REGION Network 97: ---
   RUNG wire#powerrail
      Contact( "ON" )
      wire#w1
      Contact( #FB_Enfardadora.EnPaletizadoUT )
      Contact( #Ordenes.TElev_Enfradar )
      wire#w2
      S_Coil( #FB_Enfardadora.ConEnfardadoUT )
   END_RUNG
   RUNG wire#w2
      R_Coil( #FB_Enfardadora.SinEnfardadoUT )
   END_RUNG
   RUNG wire#w1
      I_Contact( #FB_Enfardadora.EnPaletizadoUT )
      wire#w3
      R_Coil( #FB_Enfardadora.ConEnfardadoUT )
   END_RUNG
   RUNG wire#w3
      R_Coil( #FB_Enfardadora.SinEnfardadoUT )
   END_RUNG
   // the same network as SCL:
   IF "ON" AND #FB_Enfardadora.EnPaletizadoUT AND #Ordenes.TElev_Enfradar THEN
       #FB_Enfardadora.ConEnfardadoUT := TRUE;
       #FB_Enfardadora.SinEnfardadoUT := FALSE;
   END_IF;
   IF "ON" AND NOT #FB_Enfardadora.EnPaletizadoUT THEN
       #FB_Enfardadora.ConEnfardadoUT := FALSE;
       #FB_Enfardadora.SinEnfardadoUT := FALSE;
   END_IF;
END_REGION

NETWORK
TITLE = ---
/////////////////////////////////////////////////////////////////////////
// Estado para la Enfardadora

      L     P##EstadoZonaEnfa;  // Puntero a Estado ZONA
      T     #P_EstadoZonaEnfa;

      L     0;  // Inicilizo
      T     LW [#P_EstadoZonaEnfa];

// Automatico - Manual

      A     #EstadoZonaMesa.Automatico_CBx;
      =     #EstadoZonaEnfa.Automatico_CBx;

      A     #EstadoZonaMesa.Manual_CBx;
      =     #EstadoZonaEnfa.Manual_CBx;

// Marcha - Paro - Error

      A     #EstadoZonaMesa.Marcha_CBx;
      =     #EstadoZonaEnfa.Marcha_CBx;

      A     #EstadoZonaMesa.Paro_CBx;
      =     #EstadoZonaEnfa.Paro_CBx;

      A     #EstadoZonaMesa.Error_CBx;
      O     #EstadoZonaMaquina.Error_CBx;
      =     #EstadoZonaEnfa.Error_CBx;

// Reset

      A     #EstadoZonaMesa.Resetear_CBx;
      =     #EstadoZonaEnfa.Resetear_CBx;


REGION Network 99: ---
   RUNG wire#powerrail
      I_Contact( #DesHabilitar_Enfadadora )
      #FB_Enfardadora(CheckElev_EnEnfardadora := wire#w1, EstadoZona := #EstadoZonaEnfa, NDB_Enfardadora := #NDB_Enfardadora, NumMaquina := #MesaElevador, PosicionActual := #PosicionActual, DesHabitar_Enfa := #DesHabilitar_Enfadadora, PorCapas_Enfa := #PorCapas_Enfardado)
   END_RUNG
   RUNG wire#powerrail
      Contact( #CheckElev_EnEnfardadora )
   END_RUNG wire#w1
   RUNG wire#powerrail
      Contact( #ReferenciaOK_Elev )
      { S7_Templates := "SrcType := Int" } LE_Contact(in1 := #PosicionActual, in2 := #PosicionEnfardado)
   END_RUNG wire#w1
   // the same network as SCL:
   IF NOT #DesHabilitar_Enfadadora THEN
       #FB_Enfardadora(EstadoZona := #EstadoZonaEnfa,   // "FB384_Enfardadora_Paletizador_NDD"
                       NDB_Enfardadora := #NDB_Enfardadora,
                       NumMaquina := #MesaElevador,
                       PosicionActual := #PosicionActual,
                       DesHabitar_Enfa := #DesHabilitar_Enfadadora,
                       PorCapas_Enfa := #PorCapas_Enfardado,
                       CheckElev_EnEnfardadora := #CheckElev_EnEnfardadora OR (#ReferenciaOK_Elev AND (#PosicionActual <= #PosicionEnfardado)));
   END_IF;
END_REGION

REGION Network 100: Eventos de Paletizado: Inicio
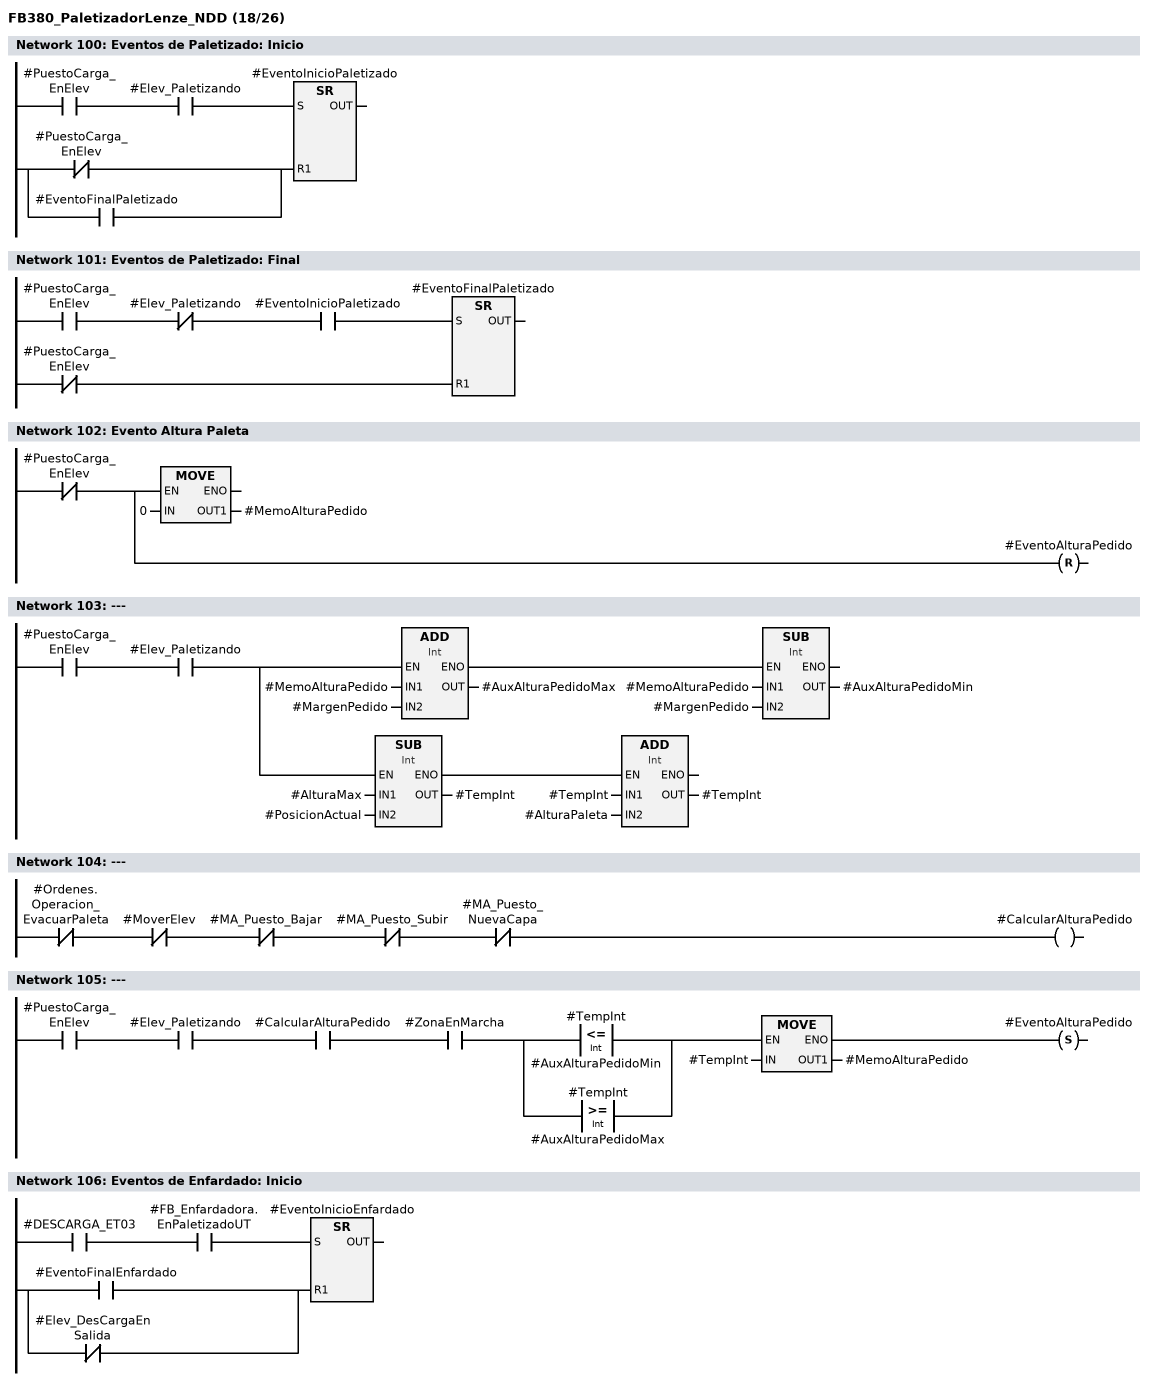
   RUNG wire#powerrail
      Contact( #PuestoCarga_EnElev )
      Contact( #Elev_Paletizando )
      S_SR(operand := #EventoInicioPaletizado, r1 := wire#w1)
   END_RUNG
   RUNG wire#powerrail
      I_Contact( #PuestoCarga_EnElev )
   END_RUNG wire#w1
   RUNG wire#powerrail
      Contact( #EventoFinalPaletizado )
   END_RUNG wire#w1
   // the same network as SCL:
   IF #PuestoCarga_EnElev AND #Elev_Paletizando THEN
       #EventoInicioPaletizado := TRUE;   // SR flip-flop
   END_IF;
   IF NOT #PuestoCarga_EnElev OR #EventoFinalPaletizado THEN #EventoInicioPaletizado := FALSE; END_IF;
END_REGION

REGION Network 101: Eventos de Paletizado: Final
   RUNG wire#powerrail
      Contact( #PuestoCarga_EnElev )
      I_Contact( #Elev_Paletizando )
      Contact( #EventoInicioPaletizado )
      S_SR(operand := #EventoFinalPaletizado, r1 := wire#w1)
   END_RUNG
   RUNG wire#powerrail
      I_Contact( #PuestoCarga_EnElev )
   END_RUNG wire#w1
   // the same network as SCL:
   IF #PuestoCarga_EnElev AND NOT #Elev_Paletizando AND #EventoInicioPaletizado THEN
       #EventoFinalPaletizado := TRUE;   // SR flip-flop
   END_IF;
   IF NOT #PuestoCarga_EnElev THEN #EventoFinalPaletizado := FALSE; END_IF;
END_REGION

REGION Network 102: Evento Altura Paleta
   RUNG wire#powerrail
      I_Contact( #PuestoCarga_EnElev )
      wire#w1
      { S7_GenerateENO := "TRUE" } Move(in := 0, out1 => #MemoAlturaPedido)
   END_RUNG
   RUNG wire#w1
      R_Coil( #EventoAlturaPedido )
   END_RUNG
   // the same network as SCL:
   IF NOT #PuestoCarga_EnElev THEN
       #MemoAlturaPedido := 0;
       #EventoAlturaPedido := FALSE;
   END_IF;
END_REGION

REGION Network 103: ---
   RUNG wire#powerrail
      Contact( #PuestoCarga_EnElev )
      Contact( #Elev_Paletizando )
      wire#w1
      { S7_Templates := "SrcType := Int"; S7_GenerateENO := "TRUE" } Add(in1 := #MemoAlturaPedido, in2 := #MargenPedido, out => #AuxAlturaPedidoMax)
      { S7_Templates := "SrcType := Int"; S7_GenerateENO := "TRUE" } Sub(in1 := #MemoAlturaPedido, in2 := #MargenPedido, out => #AuxAlturaPedidoMin)
   END_RUNG
   RUNG wire#w1
      { S7_Templates := "SrcType := Int"; S7_GenerateENO := "TRUE" } Sub(in1 := #AlturaMax, in2 := #PosicionActual, out => #TempInt)
      { S7_Templates := "SrcType := Int"; S7_GenerateENO := "TRUE" } Add(in1 := #TempInt, in2 := #AlturaPaleta, out => #TempInt)
   END_RUNG
   // the same network as SCL:
   // ENO of a box is taken as its EN; it also drops when the box reports an error
   IF #PuestoCarga_EnElev AND #Elev_Paletizando THEN
       #AuxAlturaPedidoMax := #MemoAlturaPedido + #MargenPedido;
       #AuxAlturaPedidoMin := #MemoAlturaPedido - #MargenPedido;
       #TempInt := #AlturaMax - #PosicionActual;
       #TempInt := #TempInt + #AlturaPaleta;
   END_IF;
END_REGION

REGION Network 104: ---
   RUNG wire#powerrail
      I_Contact( #Ordenes.Operacion_EvacuarPaleta )
      I_Contact( #MoverElev )
      I_Contact( #MA_Puesto_Bajar )
      I_Contact( #MA_Puesto_Subir )
      I_Contact( #MA_Puesto_NuevaCapa )
      Coil( #CalcularAlturaPedido )
   END_RUNG
   // the same network as SCL:
   #CalcularAlturaPedido := NOT #Ordenes.Operacion_EvacuarPaleta AND NOT #MoverElev AND NOT #MA_Puesto_Bajar AND NOT #MA_Puesto_Subir AND NOT #MA_Puesto_NuevaCapa;
END_REGION

REGION Network 105: ---
   RUNG wire#powerrail
      Contact( #PuestoCarga_EnElev )
      Contact( #Elev_Paletizando )
      Contact( #CalcularAlturaPedido )
      Contact( #ZonaEnMarcha )
      wire#w1
      { S7_Templates := "SrcType := Int" } LE_Contact(in1 := #TempInt, in2 := #AuxAlturaPedidoMin)
      wire#w2
      { S7_GenerateENO := "TRUE" } Move(in := #TempInt, out1 => #MemoAlturaPedido)
      S_Coil( #EventoAlturaPedido )
   END_RUNG
   RUNG wire#w1
      { S7_Templates := "SrcType := Int" } GE_Contact(in1 := #TempInt, in2 := #AuxAlturaPedidoMax)
   END_RUNG wire#w2
   // the same network as SCL:
   // ENO of a box is taken as its EN; it also drops when the box reports an error
   IF #PuestoCarga_EnElev AND #Elev_Paletizando AND #CalcularAlturaPedido AND #ZonaEnMarcha AND ((#TempInt <= #AuxAlturaPedidoMin) OR (#TempInt >= #AuxAlturaPedidoMax)) THEN
       #MemoAlturaPedido := #TempInt;
       #EventoAlturaPedido := TRUE;
   END_IF;
END_REGION

REGION Network 106: Eventos de Enfardado: Inicio
   RUNG wire#powerrail
      Contact( #DESCARGA_ET03 )
      Contact( #FB_Enfardadora.EnPaletizadoUT )
      S_SR(operand := #EventoInicioEnfardado, r1 := wire#w1)
   END_RUNG
   RUNG wire#powerrail
      Contact( #EventoFinalEnfardado )
   END_RUNG wire#w1
   RUNG wire#powerrail
      I_Contact( #Elev_DesCargaEnSalida )
   END_RUNG wire#w1
   // the same network as SCL:
   IF #DESCARGA_ET03 AND #FB_Enfardadora.EnPaletizadoUT THEN
       #EventoInicioEnfardado := TRUE;   // SR flip-flop
   END_IF;
   IF #EventoFinalEnfardado OR NOT #Elev_DesCargaEnSalida THEN #EventoInicioEnfardado := FALSE; END_IF;
END_REGION

REGION Network 107: Eventos de Enfardado: Final
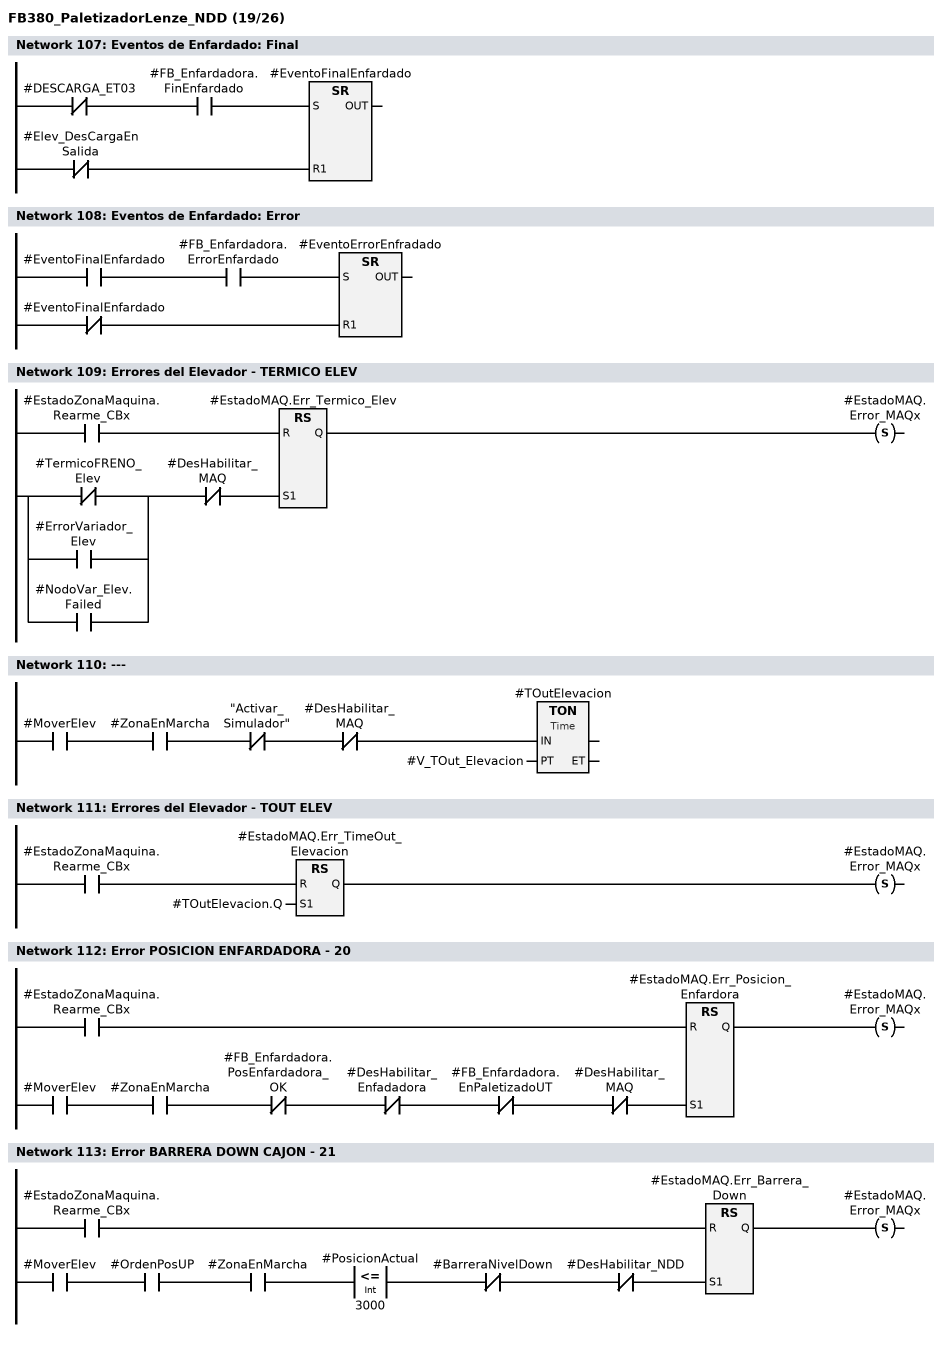
   RUNG wire#powerrail
      I_Contact( #DESCARGA_ET03 )
      Contact( #FB_Enfardadora.FinEnfardado )
      S_SR(operand := #EventoFinalEnfardado, r1 := wire#w1)
   END_RUNG
   RUNG wire#powerrail
      I_Contact( #Elev_DesCargaEnSalida )
   END_RUNG wire#w1
   // the same network as SCL:
   IF NOT #DESCARGA_ET03 AND #FB_Enfardadora.FinEnfardado THEN
       #EventoFinalEnfardado := TRUE;   // SR flip-flop
   END_IF;
   IF NOT #Elev_DesCargaEnSalida THEN #EventoFinalEnfardado := FALSE; END_IF;
END_REGION

REGION Network 108: Eventos de Enfardado: Error
   RUNG wire#powerrail
      Contact( #EventoFinalEnfardado )
      Contact( #FB_Enfardadora.ErrorEnfardado )
      S_SR(operand := #EventoErrorEnfradado, r1 := wire#w1)
   END_RUNG
   RUNG wire#powerrail
      I_Contact( #EventoFinalEnfardado )
   END_RUNG wire#w1
   // the same network as SCL:
   IF #EventoFinalEnfardado AND #FB_Enfardadora.ErrorEnfardado THEN
       #EventoErrorEnfradado := TRUE;   // SR flip-flop
   END_IF;
   IF NOT #EventoFinalEnfardado THEN #EventoErrorEnfradado := FALSE; END_IF;
END_REGION

REGION Network 109: Errores del Elevador - TERMICO ELEV
   RUNG wire#powerrail
      Contact( #EstadoZonaMaquina.Rearme_CBx )
      S_RS(operand := #EstadoMAQ.Err_Termico_Elev, s1 := wire#w2)
      S_Coil( #EstadoMAQ.Error_MAQx )
   END_RUNG
   RUNG wire#powerrail
      I_Contact( #TermicoFRENO_Elev )
      wire#w1
      I_Contact( #DesHabilitar_MAQ )
   END_RUNG wire#w2
   RUNG wire#powerrail
      Contact( #ErrorVariador_Elev )
   END_RUNG wire#w1
   RUNG wire#powerrail
      Contact( #NodoVar_Elev.Failed )
   END_RUNG wire#w1
   // the same network as SCL:
   IF #EstadoZonaMaquina.Rearme_CBx THEN
       #EstadoMAQ.Err_Termico_Elev := FALSE;   // RS flip-flop
   END_IF;
   IF (NOT #TermicoFRENO_Elev OR #ErrorVariador_Elev OR #NodoVar_Elev.Failed) AND NOT #DesHabilitar_MAQ THEN
       #EstadoMAQ.Err_Termico_Elev := TRUE;
   END_IF;
   IF #EstadoMAQ.Err_Termico_Elev THEN #EstadoMAQ.Error_MAQx := TRUE; END_IF;
END_REGION

REGION Network 110: ---
   RUNG wire#powerrail
      Contact( #MoverElev )
      Contact( #ZonaEnMarcha )
      I_Contact( "Activar_Simulador" )
      I_Contact( #DesHabilitar_MAQ )
      { S7_Templates := "time_type := Time" } #TOutElevacion.TON(pt := #V_TOut_Elevacion, et =>)
   END_RUNG
   // the same network as SCL:
   #TOutElevacion(IN := #MoverElev AND #ZonaEnMarcha AND NOT "Activar_Simulador" AND NOT #DesHabilitar_MAQ,   // TON
                  PT := #V_TOut_Elevacion);
END_REGION

REGION Network 111: Errores del Elevador - TOUT ELEV
   RUNG wire#powerrail
      Contact( #EstadoZonaMaquina.Rearme_CBx )
      S_RS(operand := #EstadoMAQ.Err_TimeOut_Elevacion, s1 := #TOutElevacion.Q)
      S_Coil( #EstadoMAQ.Error_MAQx )
   END_RUNG
   // the same network as SCL:
   IF #EstadoZonaMaquina.Rearme_CBx THEN
       #EstadoMAQ.Err_TimeOut_Elevacion := FALSE;   // RS flip-flop
   END_IF;
   IF #TOutElevacion.Q THEN #EstadoMAQ.Err_TimeOut_Elevacion := TRUE; END_IF;
   IF #EstadoMAQ.Err_TimeOut_Elevacion THEN #EstadoMAQ.Error_MAQx := TRUE; END_IF;
END_REGION

REGION Network 112: Error POSICION ENFARDADORA - 20
   RUNG wire#powerrail
      Contact( #EstadoZonaMaquina.Rearme_CBx )
      S_RS(operand := #EstadoMAQ.Err_Posicion_Enfardora, s1 := wire#w1)
      S_Coil( #EstadoMAQ.Error_MAQx )
   END_RUNG
   RUNG wire#powerrail
      Contact( #MoverElev )
      Contact( #ZonaEnMarcha )
      I_Contact( #FB_Enfardadora.PosEnfardadora_OK )
      I_Contact( #DesHabilitar_Enfadadora )
      I_Contact( #FB_Enfardadora.EnPaletizadoUT )
      I_Contact( #DesHabilitar_MAQ )
   END_RUNG wire#w1
   // the same network as SCL:
   IF #EstadoZonaMaquina.Rearme_CBx THEN
       #EstadoMAQ.Err_Posicion_Enfardora := FALSE;   // RS flip-flop
   END_IF;
   IF #MoverElev AND #ZonaEnMarcha AND NOT #FB_Enfardadora.PosEnfardadora_OK AND NOT #DesHabilitar_Enfadadora AND NOT #FB_Enfardadora.EnPaletizadoUT AND NOT #DesHabilitar_MAQ THEN
       #EstadoMAQ.Err_Posicion_Enfardora := TRUE;
   END_IF;
   IF #EstadoMAQ.Err_Posicion_Enfardora THEN #EstadoMAQ.Error_MAQx := TRUE; END_IF;
END_REGION

REGION Network 113: Error BARRERA DOWN CAJON - 21
   RUNG wire#powerrail
      Contact( #EstadoZonaMaquina.Rearme_CBx )
      S_RS(operand := #EstadoMAQ.Err_Barrera_Down, s1 := wire#w1)
      S_Coil( #EstadoMAQ.Error_MAQx )
   END_RUNG
   RUNG wire#powerrail
      Contact( #MoverElev )
      Contact( #OrdenPosUP )
      Contact( #ZonaEnMarcha )
      { S7_Templates := "SrcType := Int" } LE_Contact(in1 := #PosicionActual, in2 := 3000)
      I_Contact( #BarreraNivelDown )
      I_Contact( #DesHabilitar_NDD )
   END_RUNG wire#w1
   // the same network as SCL:
   IF #EstadoZonaMaquina.Rearme_CBx THEN
       #EstadoMAQ.Err_Barrera_Down := FALSE;   // RS flip-flop
   END_IF;
   IF #MoverElev AND #OrdenPosUP AND #ZonaEnMarcha AND (#PosicionActual <= 3000) AND NOT #BarreraNivelDown AND NOT #DesHabilitar_NDD THEN
       #EstadoMAQ.Err_Barrera_Down := TRUE;
   END_IF;
   IF #EstadoMAQ.Err_Barrera_Down THEN #EstadoMAQ.Error_MAQx := TRUE; END_IF;
END_REGION

REGION Network 114: ---
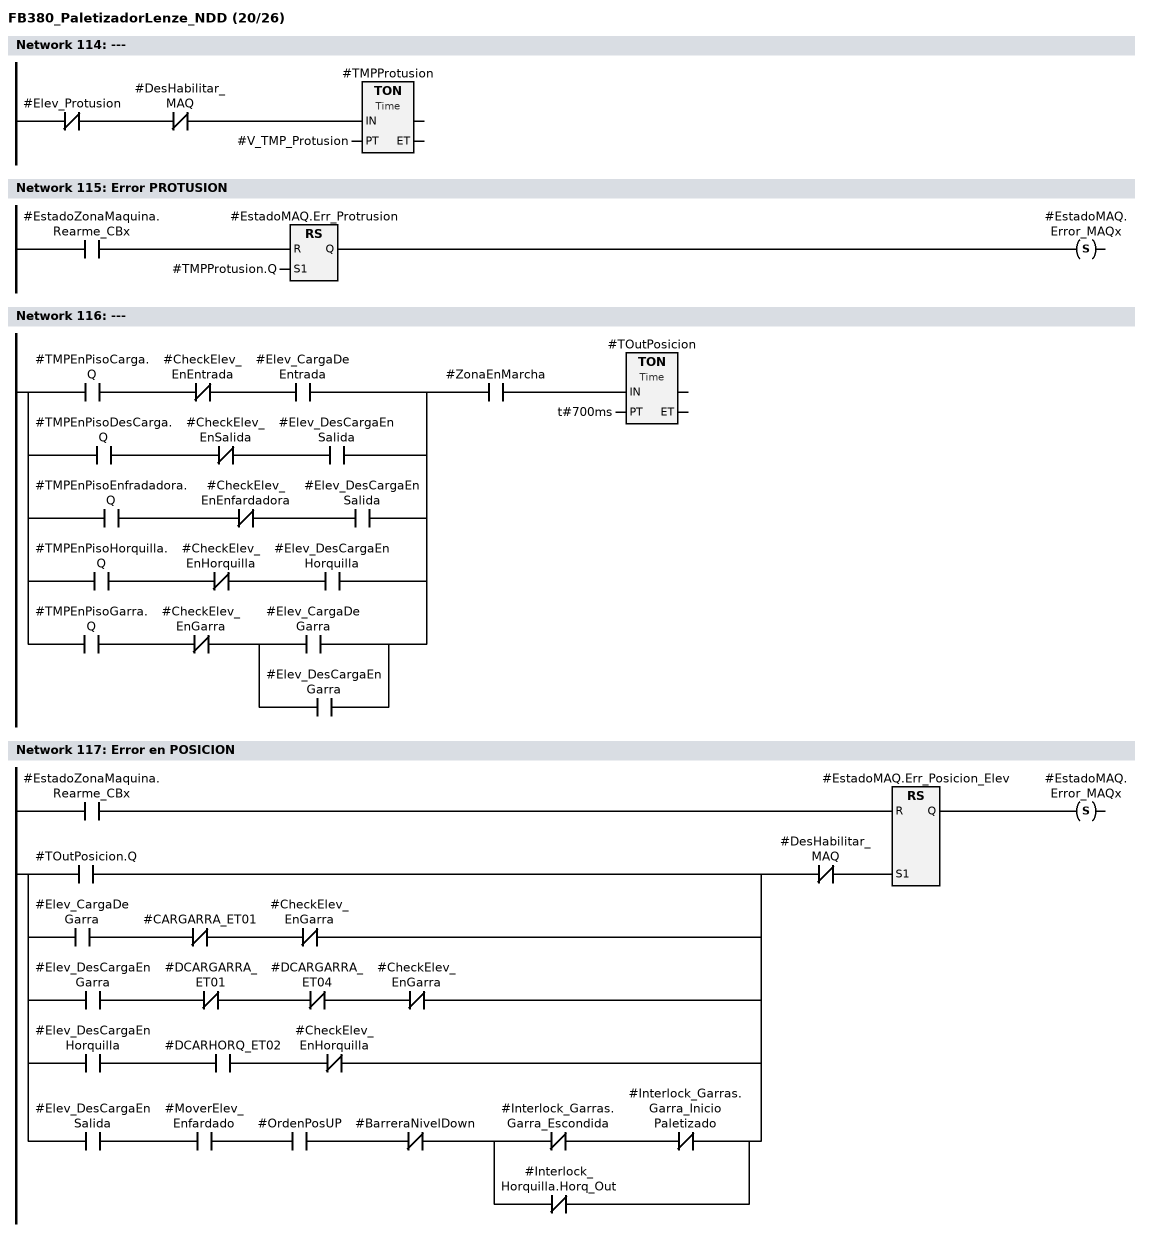
   RUNG wire#powerrail
      I_Contact( #Elev_Protusion )
      I_Contact( #DesHabilitar_MAQ )
      { S7_Templates := "time_type := Time" } #TMPProtusion.TON(pt := #V_TMP_Protusion, et =>)
   END_RUNG
   // the same network as SCL:
   #TMPProtusion(IN := NOT #Elev_Protusion AND NOT #DesHabilitar_MAQ, PT := #V_TMP_Protusion);   // TON
END_REGION

REGION Network 115: Error PROTUSION
   RUNG wire#powerrail
      Contact( #EstadoZonaMaquina.Rearme_CBx )
      S_RS(operand := #EstadoMAQ.Err_Protrusion, s1 := #TMPProtusion.Q)
      S_Coil( #EstadoMAQ.Error_MAQx )
   END_RUNG
   // the same network as SCL:
   IF #EstadoZonaMaquina.Rearme_CBx THEN
       #EstadoMAQ.Err_Protrusion := FALSE;   // RS flip-flop
   END_IF;
   IF #TMPProtusion.Q THEN #EstadoMAQ.Err_Protrusion := TRUE; END_IF;
   IF #EstadoMAQ.Err_Protrusion THEN #EstadoMAQ.Error_MAQx := TRUE; END_IF;
END_REGION

REGION Network 116: ---
   RUNG wire#powerrail
      Contact( #TMPEnPisoCarga.Q )
      I_Contact( #CheckElev_EnEntrada )
      Contact( #Elev_CargaDeEntrada )
      wire#w1
      Contact( #ZonaEnMarcha )
      { S7_Templates := "time_type := Time" } #TOutPosicion.TON(pt := t#700ms, et =>)
   END_RUNG
   RUNG wire#powerrail
      Contact( #TMPEnPisoDesCarga.Q )
      I_Contact( #CheckElev_EnSalida )
      Contact( #Elev_DesCargaEnSalida )
   END_RUNG wire#w1
   RUNG wire#powerrail
      Contact( #TMPEnPisoEnfradadora.Q )
      I_Contact( #CheckElev_EnEnfardadora )
      Contact( #Elev_DesCargaEnSalida )
   END_RUNG wire#w1
   RUNG wire#powerrail
      Contact( #TMPEnPisoHorquilla.Q )
      I_Contact( #CheckElev_EnHorquilla )
      Contact( #Elev_DesCargaEnHorquilla )
   END_RUNG wire#w1
   RUNG wire#powerrail
      Contact( #TMPEnPisoGarra.Q )
      I_Contact( #CheckElev_EnGarra )
      wire#w2
      Contact( #Elev_CargaDeGarra )
   END_RUNG wire#w1
   RUNG wire#w2
      Contact( #Elev_DesCargaEnGarra )
   END_RUNG wire#w1
   // the same network as SCL:
   #TOutPosicion(IN := ((#TMPEnPisoCarga.Q AND NOT #CheckElev_EnEntrada AND #Elev_CargaDeEntrada) OR (#TMPEnPisoDesCarga.Q AND NOT #CheckElev_EnSalida AND #Elev_DesCargaEnSalida) OR (#TMPEnPisoEnfradadora.Q AND NOT #CheckElev_EnEnfardadora AND #Elev_DesCargaEnSalida) OR (#TMPEnPisoHorquilla.Q AND NOT #CheckElev_EnHorquilla AND #Elev_DesCargaEnHorquilla) OR (#TMPEnPisoGarra.Q AND NOT #CheckElev_EnGarra AND (#Elev_CargaDeGarra OR #Elev_DesCargaEnGarra))) AND #ZonaEnMarcha,   // TON
                 PT := t#700ms);
END_REGION

REGION Network 117: Error en POSICION
   RUNG wire#powerrail
      Contact( #EstadoZonaMaquina.Rearme_CBx )
      S_RS(operand := #EstadoMAQ.Err_Posicion_Elev, s1 := wire#w3)
      S_Coil( #EstadoMAQ.Error_MAQx )
   END_RUNG
   RUNG wire#powerrail
      Contact( #TOutPosicion.Q )
      wire#w1
      I_Contact( #DesHabilitar_MAQ )
   END_RUNG wire#w3
   RUNG wire#powerrail
      Contact( #Elev_CargaDeGarra )
      I_Contact( #CARGARRA_ET01 )
      I_Contact( #CheckElev_EnGarra )
   END_RUNG wire#w1
   RUNG wire#powerrail
      Contact( #Elev_DesCargaEnGarra )
      I_Contact( #DCARGARRA_ET01 )
      I_Contact( #DCARGARRA_ET04 )
      I_Contact( #CheckElev_EnGarra )
   END_RUNG wire#w1
   RUNG wire#powerrail
      Contact( #Elev_DesCargaEnHorquilla )
      Contact( #DCARHORQ_ET02 )
      I_Contact( #CheckElev_EnHorquilla )
   END_RUNG wire#w1
   RUNG wire#powerrail
      Contact( #Elev_DesCargaEnSalida )
      Contact( #MoverElev_Enfardado )
      Contact( #OrdenPosUP )
      I_Contact( #BarreraNivelDown )
      wire#w2
      I_Contact( #Interlock_Garras.Garra_Escondida )
      I_Contact( #Interlock_Garras.Garra_InicioPaletizado )
   END_RUNG wire#w1
   RUNG wire#w2
      I_Contact( #Interlock_Horquilla.Horq_Out )
   END_RUNG wire#w1
   // the same network as SCL:
   IF #EstadoZonaMaquina.Rearme_CBx THEN
       #EstadoMAQ.Err_Posicion_Elev := FALSE;   // RS flip-flop
   END_IF;
   IF (#TOutPosicion.Q OR (#Elev_CargaDeGarra AND NOT #CARGARRA_ET01 AND NOT #CheckElev_EnGarra) OR (#Elev_DesCargaEnGarra AND NOT #DCARGARRA_ET01 AND NOT #DCARGARRA_ET04 AND NOT #CheckElev_EnGarra) OR (#Elev_DesCargaEnHorquilla AND #DCARHORQ_ET02 AND NOT #CheckElev_EnHorquilla) OR (#Elev_DesCargaEnSalida AND #MoverElev_Enfardado AND #OrdenPosUP AND NOT #BarreraNivelDown AND ((NOT #Interlock_Garras.Garra_Escondida AND NOT #Interlock_Garras.Garra_InicioPaletizado) OR NOT #Interlock_Horquilla.Horq_Out))) AND NOT #DesHabilitar_MAQ THEN
       #EstadoMAQ.Err_Posicion_Elev := TRUE;
   END_IF;
   IF #EstadoMAQ.Err_Posicion_Elev THEN #EstadoMAQ.Error_MAQx := TRUE; END_IF;
END_REGION

REGION Network 118: Error REFERENCIA ELEV - 5
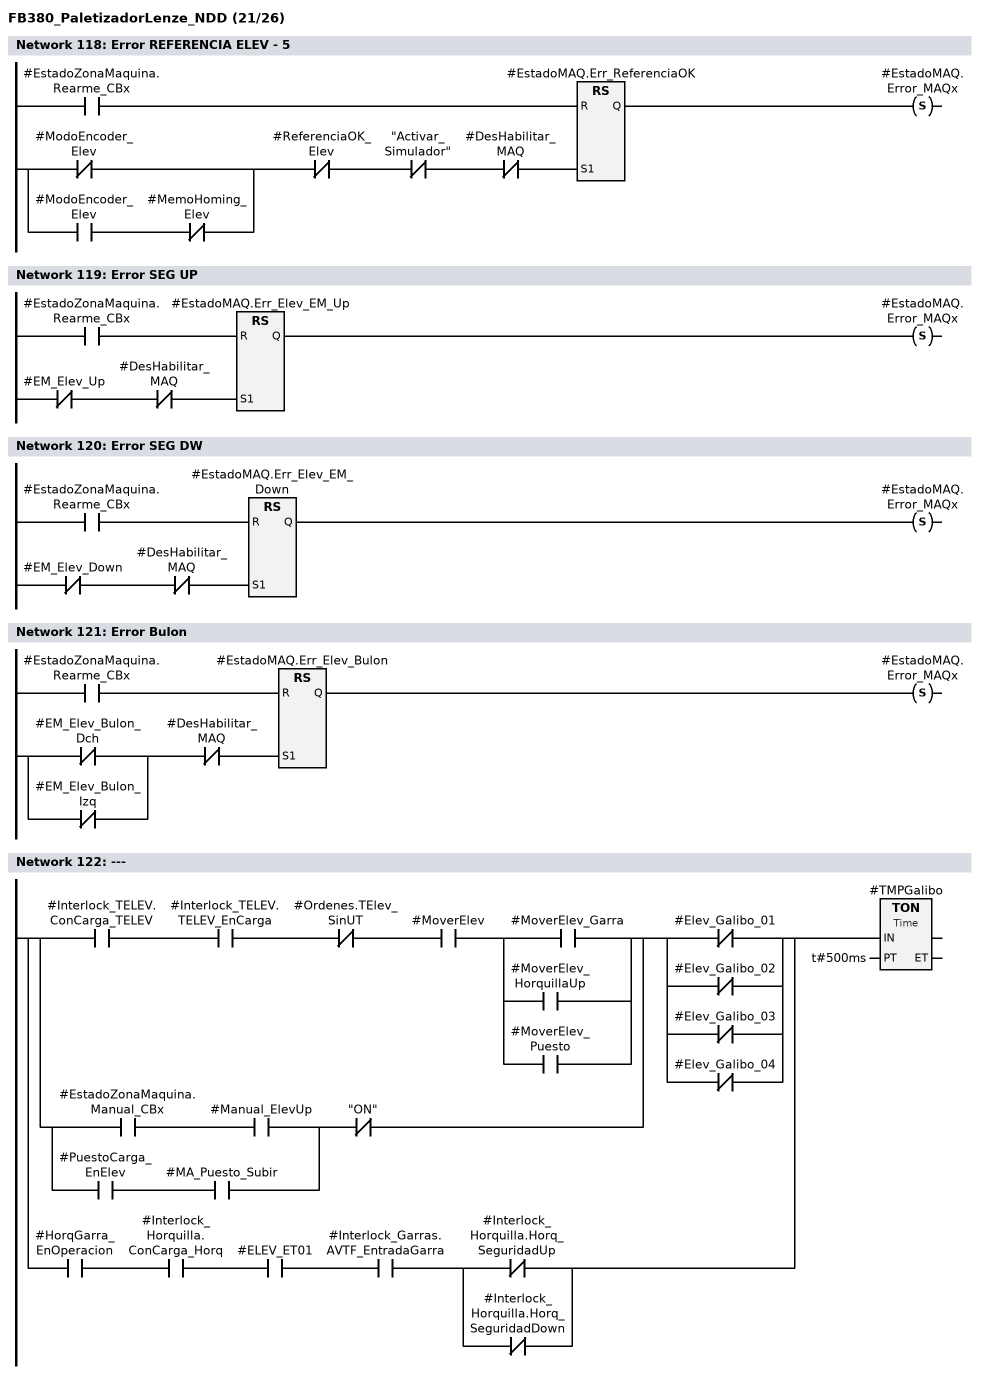
   RUNG wire#powerrail
      Contact( #EstadoZonaMaquina.Rearme_CBx )
      S_RS(operand := #EstadoMAQ.Err_ReferenciaOK, s1 := wire#w2)
      S_Coil( #EstadoMAQ.Error_MAQx )
   END_RUNG
   RUNG wire#powerrail
      I_Contact( #ModoEncoder_Elev )
      wire#w1
      I_Contact( #ReferenciaOK_Elev )
      I_Contact( "Activar_Simulador" )
      I_Contact( #DesHabilitar_MAQ )
   END_RUNG wire#w2
   RUNG wire#powerrail
      Contact( #ModoEncoder_Elev )
      I_Contact( #MemoHoming_Elev )
   END_RUNG wire#w1
   // the same network as SCL:
   IF #EstadoZonaMaquina.Rearme_CBx THEN
       #EstadoMAQ.Err_ReferenciaOK := FALSE;   // RS flip-flop
   END_IF;
   IF (NOT #ModoEncoder_Elev OR (#ModoEncoder_Elev AND NOT #MemoHoming_Elev)) AND NOT #ReferenciaOK_Elev AND NOT "Activar_Simulador" AND NOT #DesHabilitar_MAQ THEN
       #EstadoMAQ.Err_ReferenciaOK := TRUE;
   END_IF;
   IF #EstadoMAQ.Err_ReferenciaOK THEN #EstadoMAQ.Error_MAQx := TRUE; END_IF;
END_REGION

REGION Network 119: Error SEG UP
   RUNG wire#powerrail
      Contact( #EstadoZonaMaquina.Rearme_CBx )
      S_RS(operand := #EstadoMAQ.Err_Elev_EM_Up, s1 := wire#w1)
      S_Coil( #EstadoMAQ.Error_MAQx )
   END_RUNG
   RUNG wire#powerrail
      I_Contact( #EM_Elev_Up )
      I_Contact( #DesHabilitar_MAQ )
   END_RUNG wire#w1
   // the same network as SCL:
   IF #EstadoZonaMaquina.Rearme_CBx THEN
       #EstadoMAQ.Err_Elev_EM_Up := FALSE;   // RS flip-flop
   END_IF;
   IF NOT #EM_Elev_Up AND NOT #DesHabilitar_MAQ THEN #EstadoMAQ.Err_Elev_EM_Up := TRUE; END_IF;
   IF #EstadoMAQ.Err_Elev_EM_Up THEN #EstadoMAQ.Error_MAQx := TRUE; END_IF;
END_REGION

REGION Network 120: Error SEG DW
   RUNG wire#powerrail
      Contact( #EstadoZonaMaquina.Rearme_CBx )
      S_RS(operand := #EstadoMAQ.Err_Elev_EM_Down, s1 := wire#w1)
      S_Coil( #EstadoMAQ.Error_MAQx )
   END_RUNG
   RUNG wire#powerrail
      I_Contact( #EM_Elev_Down )
      I_Contact( #DesHabilitar_MAQ )
   END_RUNG wire#w1
   // the same network as SCL:
   IF #EstadoZonaMaquina.Rearme_CBx THEN
       #EstadoMAQ.Err_Elev_EM_Down := FALSE;   // RS flip-flop
   END_IF;
   IF NOT #EM_Elev_Down AND NOT #DesHabilitar_MAQ THEN #EstadoMAQ.Err_Elev_EM_Down := TRUE; END_IF;
   IF #EstadoMAQ.Err_Elev_EM_Down THEN #EstadoMAQ.Error_MAQx := TRUE; END_IF;
END_REGION

REGION Network 121: Error Bulon
   RUNG wire#powerrail
      Contact( #EstadoZonaMaquina.Rearme_CBx )
      S_RS(operand := #EstadoMAQ.Err_Elev_Bulon, s1 := wire#w2)
      S_Coil( #EstadoMAQ.Error_MAQx )
   END_RUNG
   RUNG wire#powerrail
      I_Contact( #EM_Elev_Bulon_Dch )
      wire#w1
      I_Contact( #DesHabilitar_MAQ )
   END_RUNG wire#w2
   RUNG wire#powerrail
      I_Contact( #EM_Elev_Bulon_Izq )
   END_RUNG wire#w1
   // the same network as SCL:
   IF #EstadoZonaMaquina.Rearme_CBx THEN
       #EstadoMAQ.Err_Elev_Bulon := FALSE;   // RS flip-flop
   END_IF;
   IF (NOT #EM_Elev_Bulon_Dch OR NOT #EM_Elev_Bulon_Izq) AND NOT #DesHabilitar_MAQ THEN
       #EstadoMAQ.Err_Elev_Bulon := TRUE;
   END_IF;
   IF #EstadoMAQ.Err_Elev_Bulon THEN #EstadoMAQ.Error_MAQx := TRUE; END_IF;
END_REGION

REGION Network 122: ---
   RUNG wire#powerrail
      Contact( #Interlock_TELEV.ConCarga_TELEV )
      Contact( #Interlock_TELEV.TELEV_EnCarga )
      I_Contact( #Ordenes.TElev_SinUT )
      Contact( #MoverElev )
      wire#w1
      Contact( #MoverElev_Garra )
      wire#w2
      I_Contact( #Elev_Galibo_01 )
      wire#w4
      { S7_Templates := "time_type := Time" } #TMPGalibo.TON(pt := t#500ms, et =>)
   END_RUNG
   RUNG wire#w1
      Contact( #MoverElev_HorquillaUp )
   END_RUNG wire#w2
   RUNG wire#w1
      Contact( #MoverElev_Puesto )
   END_RUNG wire#w2
   RUNG wire#powerrail
      Contact( #EstadoZonaMaquina.Manual_CBx )
      Contact( #Manual_ElevUp )
      wire#w3
      I_Contact( "ON" )
   END_RUNG wire#w2
   RUNG wire#powerrail
      Contact( #PuestoCarga_EnElev )
      Contact( #MA_Puesto_Subir )
   END_RUNG wire#w3
   RUNG wire#w2
      I_Contact( #Elev_Galibo_02 )
   END_RUNG wire#w4
   RUNG wire#w2
      I_Contact( #Elev_Galibo_03 )
   END_RUNG wire#w4
   RUNG wire#w2
      I_Contact( #Elev_Galibo_04 )
   END_RUNG wire#w4
   RUNG wire#powerrail
      Contact( #HorqGarra_EnOperacion )
      Contact( #Interlock_Horquilla.ConCarga_Horq )
      Contact( #ELEV_ET01 )
      Contact( #Interlock_Garras.AVTF_EntradaGarra )
      wire#w5
      I_Contact( #Interlock_Horquilla.Horq_SeguridadUp )
   END_RUNG wire#w4
   RUNG wire#w5
      I_Contact( #Interlock_Horquilla.Horq_SeguridadDown )
   END_RUNG wire#w4
   // the same network as SCL:
   #TMPGalibo(IN := (((#Interlock_TELEV.ConCarga_TELEV AND #Interlock_TELEV.TELEV_EnCarga AND NOT #Ordenes.TElev_SinUT AND #MoverElev AND (#MoverElev_Garra OR #MoverElev_HorquillaUp OR #MoverElev_Puesto)) OR (((#EstadoZonaMaquina.Manual_CBx AND #Manual_ElevUp) OR (#PuestoCarga_EnElev AND #MA_Puesto_Subir)) AND NOT "ON")) AND (NOT #Elev_Galibo_01 OR NOT #Elev_Galibo_02 OR NOT #Elev_Galibo_03 OR NOT #Elev_Galibo_04)) OR (#HorqGarra_EnOperacion AND #Interlock_Horquilla.ConCarga_Horq AND #ELEV_ET01 AND #Interlock_Garras.AVTF_EntradaGarra AND (NOT #Interlock_Horquilla.Horq_SeguridadUp OR NOT #Interlock_Horquilla.Horq_SeguridadDown)),   // TON
              PT := t#500ms);
END_REGION

REGION Network 123: Error PHS GALIBO
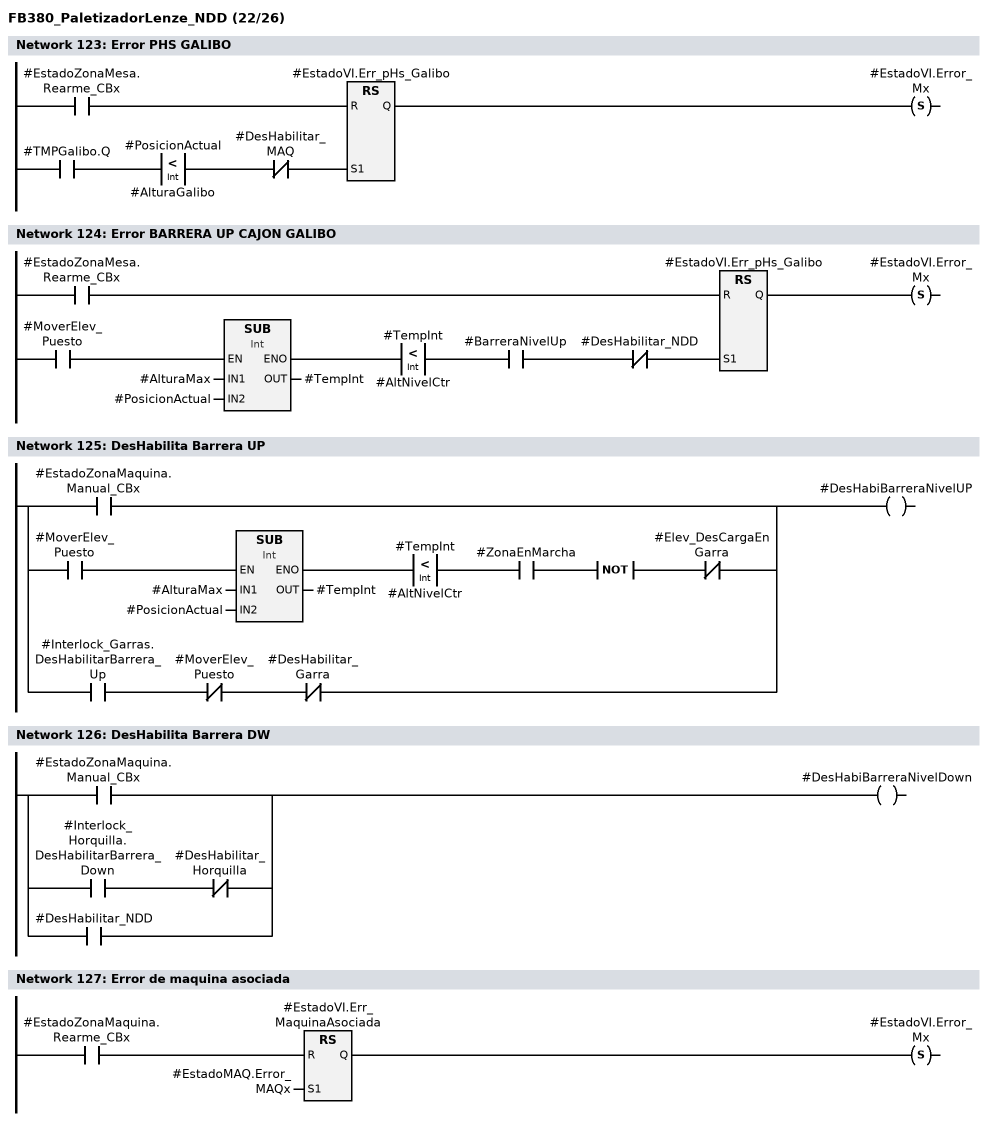
   RUNG wire#powerrail
      Contact( #EstadoZonaMesa.Rearme_CBx )
      S_RS(operand := #EstadoVI.Err_pHs_Galibo, s1 := wire#w1)
      S_Coil( #EstadoVI.Error_Mx )
   END_RUNG
   RUNG wire#powerrail
      Contact( #TMPGalibo.Q )
      { S7_Templates := "SrcType := Int" } LT_Contact(in1 := #PosicionActual, in2 := #AlturaGalibo)
      I_Contact( #DesHabilitar_MAQ )
   END_RUNG wire#w1
   // the same network as SCL:
   IF #EstadoZonaMesa.Rearme_CBx THEN
       #EstadoVI.Err_pHs_Galibo := FALSE;   // RS flip-flop
   END_IF;
   IF #TMPGalibo.Q AND (#PosicionActual < #AlturaGalibo) AND NOT #DesHabilitar_MAQ THEN
       #EstadoVI.Err_pHs_Galibo := TRUE;
   END_IF;
   IF #EstadoVI.Err_pHs_Galibo THEN #EstadoVI.Error_Mx := TRUE; END_IF;
END_REGION

REGION Network 124: Error BARRERA UP CAJON GALIBO
   RUNG wire#powerrail
      Contact( #EstadoZonaMesa.Rearme_CBx )
      S_RS(operand := #EstadoVI.Err_pHs_Galibo, s1 := wire#w1)
      S_Coil( #EstadoVI.Error_Mx )
   END_RUNG
   RUNG wire#powerrail
      Contact( #MoverElev_Puesto )
      { S7_Templates := "SrcType := Int"; S7_GenerateENO := "TRUE" } Sub(in1 := #AlturaMax, in2 := #PosicionActual, out => #TempInt)
      { S7_Templates := "SrcType := Int" } LT_Contact(in1 := #TempInt, in2 := #AltNivelCtr)
      Contact( #BarreraNivelUp )
      I_Contact( #DesHabilitar_NDD )
   END_RUNG wire#w1
   // the same network as SCL:
   // ENO of a box is taken as its EN; it also drops when the box reports an error
   IF #MoverElev_Puesto THEN #TempInt := #AlturaMax - #PosicionActual; END_IF;
   IF #EstadoZonaMesa.Rearme_CBx THEN
       #EstadoVI.Err_pHs_Galibo := FALSE;   // RS flip-flop
   END_IF;
   IF #MoverElev_Puesto AND (#TempInt < #AltNivelCtr) AND #BarreraNivelUp AND NOT #DesHabilitar_NDD THEN
       #EstadoVI.Err_pHs_Galibo := TRUE;
   END_IF;
   IF #EstadoVI.Err_pHs_Galibo THEN #EstadoVI.Error_Mx := TRUE; END_IF;
END_REGION

REGION Network 125: DesHabilita Barrera UP
   RUNG wire#powerrail
      Contact( #EstadoZonaMaquina.Manual_CBx )
      wire#w1
      Coil( #DesHabiBarreraNivelUP )
   END_RUNG
   RUNG wire#powerrail
      Contact( #MoverElev_Puesto )
      { S7_Templates := "SrcType := Int"; S7_GenerateENO := "TRUE" } Sub(in1 := #AlturaMax, in2 := #PosicionActual, out => #TempInt)
      { S7_Templates := "SrcType := Int" } LT_Contact(in1 := #TempInt, in2 := #AltNivelCtr)
      Contact( #ZonaEnMarcha )
      Not()
      I_Contact( #Elev_DesCargaEnGarra )
   END_RUNG wire#w1
   RUNG wire#powerrail
      Contact( #Interlock_Garras.DesHabilitarBarrera_Up )
      I_Contact( #MoverElev_Puesto )
      I_Contact( #DesHabilitar_Garra )
   END_RUNG wire#w1
   // the same network as SCL:
   // ENO of a box is taken as its EN; it also drops when the box reports an error
   IF #MoverElev_Puesto THEN #TempInt := #AlturaMax - #PosicionActual; END_IF;
   #DesHabiBarreraNivelUP := #EstadoZonaMaquina.Manual_CBx OR (NOT (#MoverElev_Puesto AND (#TempInt < #AltNivelCtr) AND #ZonaEnMarcha) AND NOT #Elev_DesCargaEnGarra) OR (#Interlock_Garras.DesHabilitarBarrera_Up AND NOT #MoverElev_Puesto AND NOT #DesHabilitar_Garra);
END_REGION

REGION Network 126: DesHabilita Barrera DW
   RUNG wire#powerrail
      Contact( #EstadoZonaMaquina.Manual_CBx )
      wire#w1
      Coil( #DesHabiBarreraNivelDown )
   END_RUNG
   RUNG wire#powerrail
      Contact( #Interlock_Horquilla.DesHabilitarBarrera_Down )
      I_Contact( #DesHabilitar_Horquilla )
   END_RUNG wire#w1
   RUNG wire#powerrail
      Contact( #DesHabilitar_NDD )
   END_RUNG wire#w1
   // the same network as SCL:
   #DesHabiBarreraNivelDown := #EstadoZonaMaquina.Manual_CBx OR (#Interlock_Horquilla.DesHabilitarBarrera_Down AND NOT #DesHabilitar_Horquilla) OR #DesHabilitar_NDD;
END_REGION

REGION Network 127: Error de maquina asociada
   RUNG wire#powerrail
      Contact( #EstadoZonaMaquina.Rearme_CBx )
      S_RS(operand := #EstadoVI.Err_MaquinaAsociada, s1 := #EstadoMAQ.Error_MAQx)
      S_Coil( #EstadoVI.Error_Mx )
   END_RUNG
   // the same network as SCL:
   IF #EstadoZonaMaquina.Rearme_CBx THEN
       #EstadoVI.Err_MaquinaAsociada := FALSE;   // RS flip-flop
   END_IF;
   IF #EstadoMAQ.Error_MAQx THEN #EstadoVI.Err_MaquinaAsociada := TRUE; END_IF;
   IF #EstadoVI.Err_MaquinaAsociada THEN #EstadoVI.Error_Mx := TRUE; END_IF;
END_REGION

REGION Network 128: Estado del Elevador
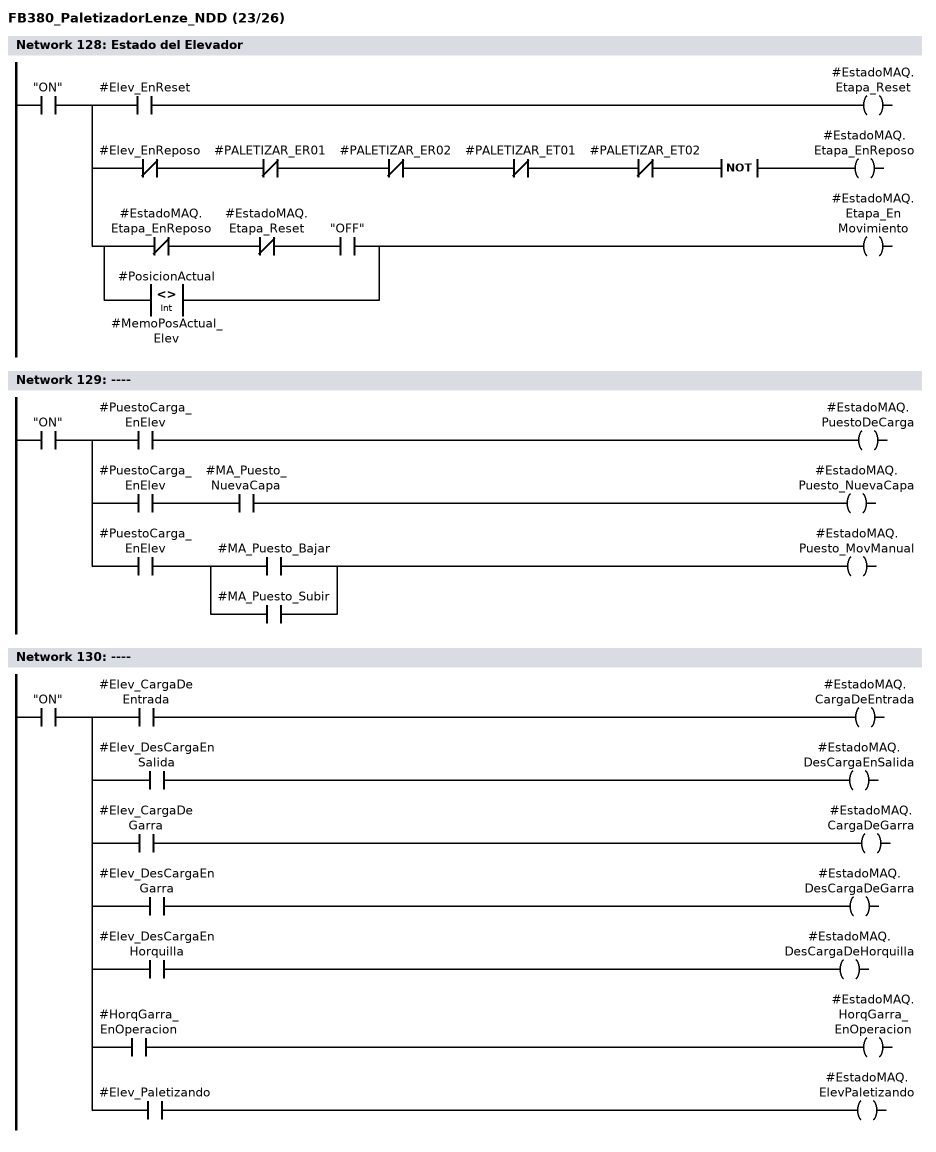
   RUNG wire#powerrail
      Contact( "ON" )
      wire#w1
      Contact( #Elev_EnReset )
      Coil( #EstadoMAQ.Etapa_Reset )
   END_RUNG
   RUNG wire#w1
      I_Contact( #Elev_EnReposo )
      I_Contact( #PALETIZAR_ER01 )
      I_Contact( #PALETIZAR_ER02 )
      I_Contact( #PALETIZAR_ET01 )
      I_Contact( #PALETIZAR_ET02 )
      Not()
      Coil( #EstadoMAQ.Etapa_EnReposo )
   END_RUNG
   RUNG wire#w1
      I_Contact( #EstadoMAQ.Etapa_EnReposo )
      I_Contact( #EstadoMAQ.Etapa_Reset )
      Contact( "OFF" )
      wire#w2
      Coil( #EstadoMAQ.Etapa_EnMovimiento )
   END_RUNG
   RUNG wire#w1
      { S7_Templates := "SrcType := Int" } NE_Contact(in1 := #PosicionActual, in2 := #MemoPosActual_Elev)
   END_RUNG wire#w2
   // the same network as SCL:
   #EstadoMAQ.Etapa_Reset := "ON" AND #Elev_EnReset;
   #EstadoMAQ.Etapa_EnReposo := NOT ("ON" AND NOT #Elev_EnReposo AND NOT #PALETIZAR_ER01 AND NOT #PALETIZAR_ER02 AND NOT #PALETIZAR_ET01 AND NOT #PALETIZAR_ET02);
   #EstadoMAQ.Etapa_EnMovimiento := "ON" AND ((NOT #EstadoMAQ.Etapa_EnReposo AND NOT #EstadoMAQ.Etapa_Reset AND "OFF") OR (#PosicionActual <> #MemoPosActual_Elev));
END_REGION

REGION Network 129: ----
   RUNG wire#powerrail
      Contact( "ON" )
      wire#w1
      Contact( #PuestoCarga_EnElev )
      Coil( #EstadoMAQ.PuestoDeCarga )
   END_RUNG
   RUNG wire#w1
      Contact( #PuestoCarga_EnElev )
      Contact( #MA_Puesto_NuevaCapa )
      Coil( #EstadoMAQ.Puesto_NuevaCapa )
   END_RUNG
   RUNG wire#w1
      Contact( #PuestoCarga_EnElev )
      wire#w2
      Contact( #MA_Puesto_Bajar )
      wire#w3
      Coil( #EstadoMAQ.Puesto_MovManual )
   END_RUNG
   RUNG wire#w2
      Contact( #MA_Puesto_Subir )
   END_RUNG wire#w3
   // the same network as SCL:
   #EstadoMAQ.PuestoDeCarga := "ON" AND #PuestoCarga_EnElev;
   #EstadoMAQ.Puesto_NuevaCapa := "ON" AND #PuestoCarga_EnElev AND #MA_Puesto_NuevaCapa;
   #EstadoMAQ.Puesto_MovManual := "ON" AND #PuestoCarga_EnElev AND (#MA_Puesto_Bajar OR #MA_Puesto_Subir);
END_REGION

REGION Network 130: ----
   RUNG wire#powerrail
      Contact( "ON" )
      wire#w1
      Contact( #Elev_CargaDeEntrada )
      Coil( #EstadoMAQ.CargaDeEntrada )
   END_RUNG
   RUNG wire#w1
      Contact( #Elev_DesCargaEnSalida )
      Coil( #EstadoMAQ.DesCargaEnSalida )
   END_RUNG
   RUNG wire#w1
      Contact( #Elev_CargaDeGarra )
      Coil( #EstadoMAQ.CargaDeGarra )
   END_RUNG
   RUNG wire#w1
      Contact( #Elev_DesCargaEnGarra )
      Coil( #EstadoMAQ.DesCargaDeGarra )
   END_RUNG
   RUNG wire#w1
      Contact( #Elev_DesCargaEnHorquilla )
      Coil( #EstadoMAQ.DesCargaDeHorquilla )
   END_RUNG
   RUNG wire#w1
      Contact( #HorqGarra_EnOperacion )
      Coil( #EstadoMAQ.HorqGarra_EnOperacion )
   END_RUNG
   RUNG wire#w1
      Contact( #Elev_Paletizando )
      Coil( #EstadoMAQ.ElevPaletizando )
   END_RUNG
   // the same network as SCL:
   #EstadoMAQ.CargaDeEntrada := "ON" AND #Elev_CargaDeEntrada;
   #EstadoMAQ.DesCargaEnSalida := "ON" AND #Elev_DesCargaEnSalida;
   #EstadoMAQ.CargaDeGarra := "ON" AND #Elev_CargaDeGarra;
   #EstadoMAQ.DesCargaDeGarra := "ON" AND #Elev_DesCargaEnGarra;
   #EstadoMAQ.DesCargaDeHorquilla := "ON" AND #Elev_DesCargaEnHorquilla;
   #EstadoMAQ.HorqGarra_EnOperacion := "ON" AND #HorqGarra_EnOperacion;
   #EstadoMAQ.ElevPaletizando := "ON" AND #Elev_Paletizando;
END_REGION

REGION Network 131: Entradas del Elevador
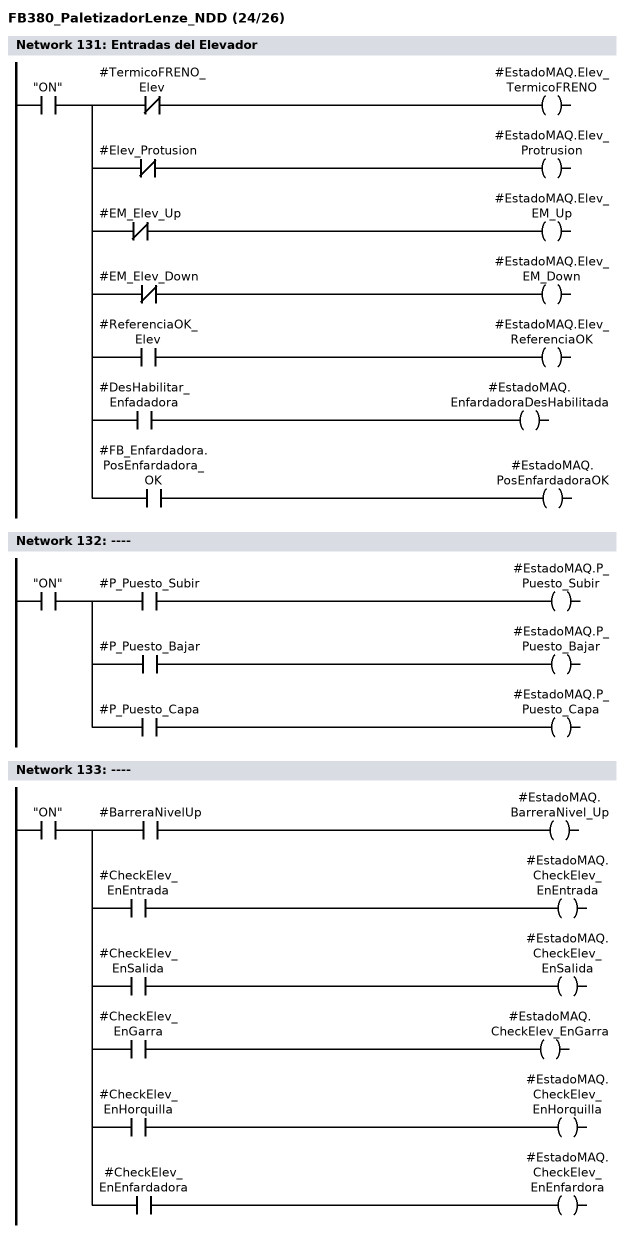
   RUNG wire#powerrail
      Contact( "ON" )
      wire#w1
      I_Contact( #TermicoFRENO_Elev )
      Coil( #EstadoMAQ.Elev_TermicoFRENO )
   END_RUNG
   RUNG wire#w1
      I_Contact( #Elev_Protusion )
      Coil( #EstadoMAQ.Elev_Protrusion )
   END_RUNG
   RUNG wire#w1
      I_Contact( #EM_Elev_Up )
      Coil( #EstadoMAQ.Elev_EM_Up )
   END_RUNG
   RUNG wire#w1
      I_Contact( #EM_Elev_Down )
      Coil( #EstadoMAQ.Elev_EM_Down )
   END_RUNG
   RUNG wire#w1
      Contact( #ReferenciaOK_Elev )
      Coil( #EstadoMAQ.Elev_ReferenciaOK )
   END_RUNG
   RUNG wire#w1
      Contact( #DesHabilitar_Enfadadora )
      Coil( #EstadoMAQ.EnfardadoraDesHabilitada )
   END_RUNG
   RUNG wire#w1
      Contact( #FB_Enfardadora.PosEnfardadora_OK )
      Coil( #EstadoMAQ.PosEnfardadoraOK )
   END_RUNG
   // the same network as SCL:
   #EstadoMAQ.Elev_TermicoFRENO := "ON" AND NOT #TermicoFRENO_Elev;
   #EstadoMAQ.Elev_Protrusion := "ON" AND NOT #Elev_Protusion;
   #EstadoMAQ.Elev_EM_Up := "ON" AND NOT #EM_Elev_Up;
   #EstadoMAQ.Elev_EM_Down := "ON" AND NOT #EM_Elev_Down;
   #EstadoMAQ.Elev_ReferenciaOK := "ON" AND #ReferenciaOK_Elev;
   #EstadoMAQ.EnfardadoraDesHabilitada := "ON" AND #DesHabilitar_Enfadadora;
   #EstadoMAQ.PosEnfardadoraOK := "ON" AND #FB_Enfardadora.PosEnfardadora_OK;
END_REGION

REGION Network 132: ----
   RUNG wire#powerrail
      Contact( "ON" )
      wire#w1
      Contact( #P_Puesto_Subir )
      Coil( #EstadoMAQ.P_Puesto_Subir )
   END_RUNG
   RUNG wire#w1
      Contact( #P_Puesto_Bajar )
      Coil( #EstadoMAQ.P_Puesto_Bajar )
   END_RUNG
   RUNG wire#w1
      Contact( #P_Puesto_Capa )
      Coil( #EstadoMAQ.P_Puesto_Capa )
   END_RUNG
   // the same network as SCL:
   #EstadoMAQ.P_Puesto_Subir := "ON" AND #P_Puesto_Subir;
   #EstadoMAQ.P_Puesto_Bajar := "ON" AND #P_Puesto_Bajar;
   #EstadoMAQ.P_Puesto_Capa := "ON" AND #P_Puesto_Capa;
END_REGION

REGION Network 133: ----
   RUNG wire#powerrail
      Contact( "ON" )
      wire#w1
      Contact( #BarreraNivelUp )
      Coil( #EstadoMAQ.BarreraNivel_Up )
   END_RUNG
   RUNG wire#w1
      Contact( #CheckElev_EnEntrada )
      Coil( #EstadoMAQ.CheckElev_EnEntrada )
   END_RUNG
   RUNG wire#w1
      Contact( #CheckElev_EnSalida )
      Coil( #EstadoMAQ.CheckElev_EnSalida )
   END_RUNG
   RUNG wire#w1
      Contact( #CheckElev_EnGarra )
      Coil( #EstadoMAQ.CheckElev_EnGarra )
   END_RUNG
   RUNG wire#w1
      Contact( #CheckElev_EnHorquilla )
      Coil( #EstadoMAQ.CheckElev_EnHorquilla )
   END_RUNG
   RUNG wire#w1
      Contact( #CheckElev_EnEnfardadora )
      Coil( #EstadoMAQ.CheckElev_EnEnfardora )
   END_RUNG
   // the same network as SCL:
   #EstadoMAQ.BarreraNivel_Up := "ON" AND #BarreraNivelUp;
   #EstadoMAQ.CheckElev_EnEntrada := "ON" AND #CheckElev_EnEntrada;
   #EstadoMAQ.CheckElev_EnSalida := "ON" AND #CheckElev_EnSalida;
   #EstadoMAQ.CheckElev_EnGarra := "ON" AND #CheckElev_EnGarra;
   #EstadoMAQ.CheckElev_EnHorquilla := "ON" AND #CheckElev_EnHorquilla;
   #EstadoMAQ.CheckElev_EnEnfardora := "ON" AND #CheckElev_EnEnfardadora;
END_REGION

REGION Network 134: ----
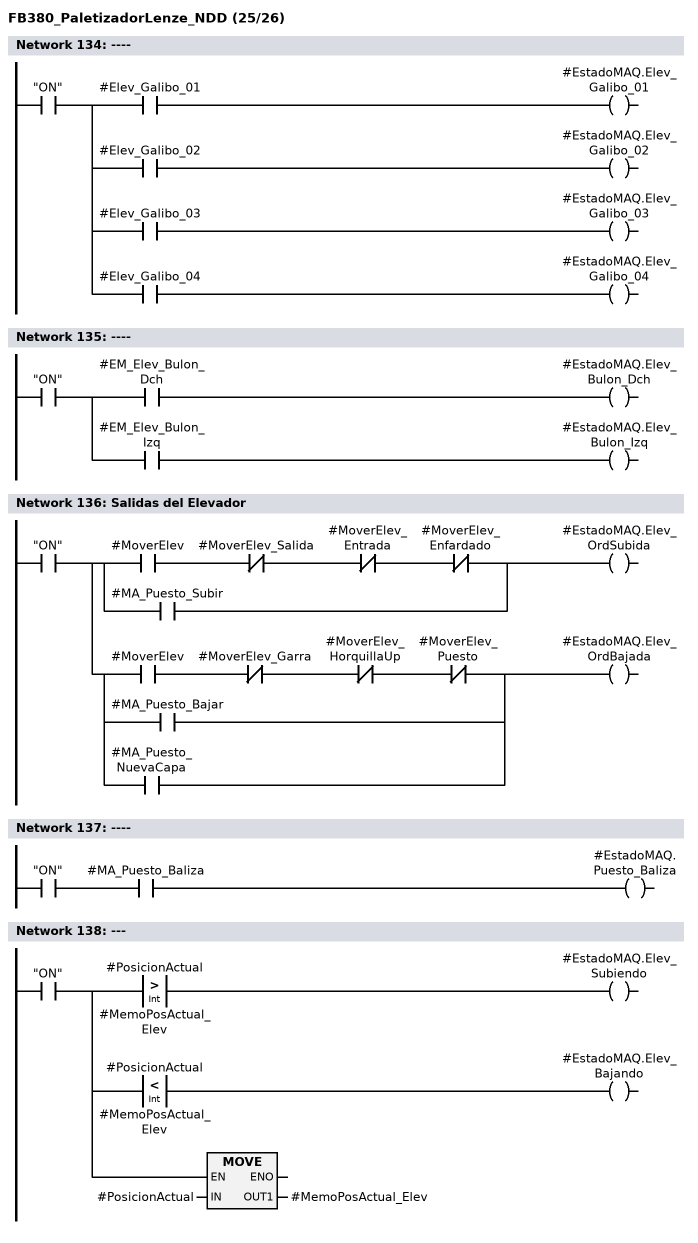
   RUNG wire#powerrail
      Contact( "ON" )
      wire#w1
      Contact( #Elev_Galibo_01 )
      Coil( #EstadoMAQ.Elev_Galibo_01 )
   END_RUNG
   RUNG wire#w1
      Contact( #Elev_Galibo_02 )
      Coil( #EstadoMAQ.Elev_Galibo_02 )
   END_RUNG
   RUNG wire#w1
      Contact( #Elev_Galibo_03 )
      Coil( #EstadoMAQ.Elev_Galibo_03 )
   END_RUNG
   RUNG wire#w1
      Contact( #Elev_Galibo_04 )
      Coil( #EstadoMAQ.Elev_Galibo_04 )
   END_RUNG
   // the same network as SCL:
   #EstadoMAQ.Elev_Galibo_01 := "ON" AND #Elev_Galibo_01;
   #EstadoMAQ.Elev_Galibo_02 := "ON" AND #Elev_Galibo_02;
   #EstadoMAQ.Elev_Galibo_03 := "ON" AND #Elev_Galibo_03;
   #EstadoMAQ.Elev_Galibo_04 := "ON" AND #Elev_Galibo_04;
END_REGION

REGION Network 135: ----
   RUNG wire#powerrail
      Contact( "ON" )
      wire#w1
      Contact( #EM_Elev_Bulon_Dch )
      Coil( #EstadoMAQ.Elev_Bulon_Dch )
   END_RUNG
   RUNG wire#w1
      Contact( #EM_Elev_Bulon_Izq )
      Coil( #EstadoMAQ.Elev_Bulon_Izq )
   END_RUNG
   // the same network as SCL:
   #EstadoMAQ.Elev_Bulon_Dch := "ON" AND #EM_Elev_Bulon_Dch;
   #EstadoMAQ.Elev_Bulon_Izq := "ON" AND #EM_Elev_Bulon_Izq;
END_REGION

REGION Network 136: Salidas del Elevador
   RUNG wire#powerrail
      Contact( "ON" )
      wire#w1
      Contact( #MoverElev )
      I_Contact( #MoverElev_Salida )
      I_Contact( #MoverElev_Entrada )
      I_Contact( #MoverElev_Enfardado )
      wire#w2
      Coil( #EstadoMAQ.Elev_OrdSubida )
   END_RUNG
   RUNG wire#w1
      Contact( #MA_Puesto_Subir )
   END_RUNG wire#w2
   RUNG wire#w1
      Contact( #MoverElev )
      I_Contact( #MoverElev_Garra )
      I_Contact( #MoverElev_HorquillaUp )
      I_Contact( #MoverElev_Puesto )
      wire#w3
      Coil( #EstadoMAQ.Elev_OrdBajada )
   END_RUNG
   RUNG wire#w1
      Contact( #MA_Puesto_Bajar )
   END_RUNG wire#w3
   RUNG wire#w1
      Contact( #MA_Puesto_NuevaCapa )
   END_RUNG wire#w3
   // the same network as SCL:
   #EstadoMAQ.Elev_OrdSubida := "ON" AND ((#MoverElev AND NOT #MoverElev_Salida AND NOT #MoverElev_Entrada AND NOT #MoverElev_Enfardado) OR #MA_Puesto_Subir);
   #EstadoMAQ.Elev_OrdBajada := "ON" AND ((#MoverElev AND NOT #MoverElev_Garra AND NOT #MoverElev_HorquillaUp AND NOT #MoverElev_Puesto) OR #MA_Puesto_Bajar OR #MA_Puesto_NuevaCapa);
END_REGION

REGION Network 137: ----
   RUNG wire#powerrail
      Contact( "ON" )
      Contact( #MA_Puesto_Baliza )
      Coil( #EstadoMAQ.Puesto_Baliza )
   END_RUNG
   // the same network as SCL:
   #EstadoMAQ.Puesto_Baliza := "ON" AND #MA_Puesto_Baliza;
END_REGION

REGION Network 138: ---
   RUNG wire#powerrail
      Contact( "ON" )
      wire#w1
      { S7_Templates := "SrcType := Int" } GT_Contact(in1 := #PosicionActual, in2 := #MemoPosActual_Elev)
      Coil( #EstadoMAQ.Elev_Subiendo )
   END_RUNG
   RUNG wire#w1
      { S7_Templates := "SrcType := Int" } LT_Contact(in1 := #PosicionActual, in2 := #MemoPosActual_Elev)
      Coil( #EstadoMAQ.Elev_Bajando )
   END_RUNG
   RUNG wire#w1
      { S7_GenerateENO := "TRUE" } Move(in := #PosicionActual, out1 => #MemoPosActual_Elev)
   END_RUNG
   // the same network as SCL:
   #EstadoMAQ.Elev_Subiendo := "ON" AND (#PosicionActual > #MemoPosActual_Elev);
   #EstadoMAQ.Elev_Bajando := "ON" AND (#PosicionActual < #MemoPosActual_Elev);
   IF "ON" THEN #MemoPosActual_Elev := #PosicionActual; END_IF;
END_REGION

NETWORK
TITLE = Posicion del Elevador para la pantalla
// Estado Maquina W14 reservado para la PosActual y el W10 reservado por utilizar
      L     P#0.0;
      T     #P_Temporal;  // Reiniciamos el puntero

      L     #MesaElevador;  // Numero de la maquina a copiar
      L     16;  // Tamaño de la estructura de cada maquina
      *I;
      L     14;  // Posicion de la palabra que se quierre escribir
      +I;
      SLD   3;  // Comando para pasar a formato Puntero
      T     #P_Temporal;

      OPN   "DB904_Estado_Maquinas";  // Abrimos el DB donde se va a escribir la informacion

      L     #PosicionActual;  // Cargamos la informacion
      T     DBW [#P_Temporal];  // Escribimos en la posicion indicada



REGION Network 140: Datos de la Scada
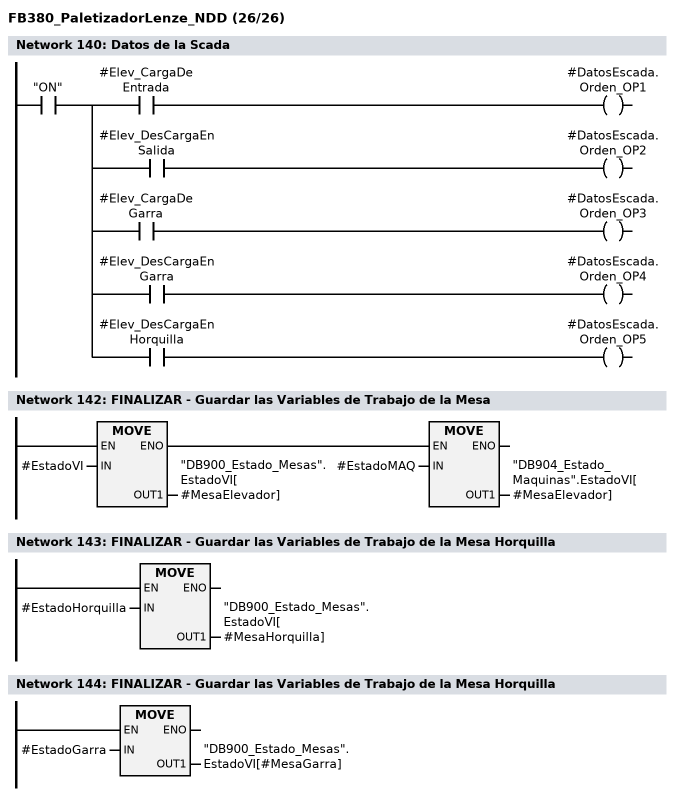
   RUNG wire#powerrail
      Contact( "ON" )
      wire#w1
      Contact( #Elev_CargaDeEntrada )
      Coil( #DatosEscada.Orden_OP1 )
   END_RUNG
   RUNG wire#w1
      Contact( #Elev_DesCargaEnSalida )
      Coil( #DatosEscada.Orden_OP2 )
   END_RUNG
   RUNG wire#w1
      Contact( #Elev_CargaDeGarra )
      Coil( #DatosEscada.Orden_OP3 )
   END_RUNG
   RUNG wire#w1
      Contact( #Elev_DesCargaEnGarra )
      Coil( #DatosEscada.Orden_OP4 )
   END_RUNG
   RUNG wire#w1
      Contact( #Elev_DesCargaEnHorquilla )
      Coil( #DatosEscada.Orden_OP5 )
   END_RUNG
   // the same network as SCL:
   #DatosEscada.Orden_OP1 := "ON" AND #Elev_CargaDeEntrada;
   #DatosEscada.Orden_OP2 := "ON" AND #Elev_DesCargaEnSalida;
   #DatosEscada.Orden_OP3 := "ON" AND #Elev_CargaDeGarra;
   #DatosEscada.Orden_OP4 := "ON" AND #Elev_DesCargaEnGarra;
   #DatosEscada.Orden_OP5 := "ON" AND #Elev_DesCargaEnHorquilla;
END_REGION

REGION Network 141: ---
END_REGION

REGION Network 142: FINALIZAR - Guardar las Variables de Trabajo de la Mesa
   RUNG wire#powerrail
      Move(in := #EstadoVI, out1 => "DB900_Estado_Mesas".EstadoVI[#MesaElevador])
      Move(in := #EstadoMAQ, out1 => "DB904_Estado_Maquinas".EstadoVI[#MesaElevador])
   END_RUNG
   // the same network as SCL:
   "DB900_Estado_Mesas".EstadoVI[#MesaElevador] := #EstadoVI;
   "DB904_Estado_Maquinas".EstadoVI[#MesaElevador] := #EstadoMAQ;
END_REGION

REGION Network 143: FINALIZAR - Guardar las Variables de Trabajo de la Mesa Horquilla
   RUNG wire#powerrail
      Move(in := #EstadoHorquilla, out1 => "DB900_Estado_Mesas".EstadoVI[#MesaHorquilla])
   END_RUNG
   // the same network as SCL:
   "DB900_Estado_Mesas".EstadoVI[#MesaHorquilla] := #EstadoHorquilla;
END_REGION

REGION Network 144: FINALIZAR - Guardar las Variables de Trabajo de la Mesa Horquilla
   RUNG wire#powerrail
      Move(in := #EstadoGarra, out1 => "DB900_Estado_Mesas".EstadoVI[#MesaGarra])
   END_RUNG
   // the same network as SCL:
   "DB900_Estado_Mesas".EstadoVI[#MesaGarra] := #EstadoGarra;
END_REGION
END_FUNCTION_BLOCK
